(* IEC 61131-3 sources: plc_simulator/services/codesys/POUs (part 11) *)

(* ---- TWA_FB_CalcLimits.st ---- *)
(* ===========================================================================================
 *  TWA_FB_CalcLimits — Transporter Working Area: X-limit calculation
 *
 *  Company : Galvatek part of the John Cockerill Group
 *  Author  : Jarmo Piipponen
 *  Created : 25.03.2026
 *
 * -------------------------------------------------------------------------------------------
 *  Calculates x_min_limit and x_max_limit for all active
 *  transporters. Collision avoidance layers:
 *
 *  Pass 1 (per transporter):
 *  - Station restrictions from g_avoid_status
 *  - Safety distance from same-line neighbors
 *  - canEvade, priority, x-rank computation
 *
 *  Pass 2 (pair comparisons):
 *  - Priority-based restrictions (higher → lower)
 *  - Bidirectional safety (same direction chase)
 *
 *  Final: Trap validation
 *
 *  ------------------------------------------------------------------------------------------
 *
 *  Changes:
 *
 *
 *
 *)

FUNCTION_BLOCK TWA_FB_CalcLimits

(* Introduction of Variables ----------------------------------------------------------------*)

VAR_EXTERNAL CONSTANT
    MAX_TRANSPORTERS        : INT;
    MAX_UNITS               : INT;
    MIN_STATION_INDEX        : INT;
    MAX_STATION_INDEX        : INT;
    AVOID_PASSABLE          : INT;
    AVOID_BLOCK             : INT;
    MIN_WORKING_AREA         : DINT;
    IN_PROCESS              : INT;
END_VAR

VAR_EXTERNAL
  Transporters                     : ARRAY[0..MAX_TRANSPORTERS] OF UDT_TransporterType;
  g_transporter             : ARRAY[1..MAX_TRANSPORTERS] OF UDT_TransporterStatusType;
  Stations                 : ARRAY[MIN_STATION_INDEX..MAX_STATION_INDEX] OF UDT_StationType;
  CountStations              : INT;
  g_avoid_status            : ARRAY[MIN_STATION_INDEX..MAX_STATION_INDEX] OF INT;
  g_station_occupancy             : ARRAY[1..MAX_STATION_INDEX] OF UDT_JC_UnitAtStationType;
  g_batch                   : ARRAY[1..MAX_UNITS] OF UDT_BatchType;
END_VAR

VAR
  i                         : INT;
  j                         : INT;
  stn_num                   : INT;
  stn_x                     : DINT;
  avoid_st                  : INT;
  min_x                     : DINT;
  max_x                     : DINT;
  current_x                 : DINT;
  current_y                 : DINT;
  avoid_dist                : DINT;
  is_target                 : BOOL;
  new_val                   : DINT;

  (* Station scan: nearest restricting station per side *)
  near_left_x               : DINT;
  near_left_stn             : INT;
  near_right_x              : DINT;
  near_right_stn            : INT;
  has_left                  : BOOL;
  has_right                 : BOOL;
  midpoint                  : DINT;

  (* Per-transporter computed values *)
  priority                  : ARRAY[1..MAX_TRANSPORTERS] OF DINT;
  can_evade                 : ARRAY[1..MAX_TRANSPORTERS] OF BOOL;
  rank                      : ARRAY[1..MAX_TRANSPORTERS] OF INT;

  (* Pair comparison *)
  other_x                   : DINT;
  other_y                   : DINT;
  i_phase                   : INT;
  j_phase                   : INT;
  dist                      : DINT;
  work_area                 : DINT;
  a_wins                    : BOOL;
  restrict_x                : DINT;
  between                   : INT;
  chain_ofs                 : DINT;
  adjusted                  : DINT;

  (* Bidirectional *)
  i_moving_right            : BOOL;
  i_moving_left             : BOOL;
  j_moving_right            : BOOL;
  j_moving_left             : BOOL;

  (* IN_PROCESS batch priority boost *)
  lift_stn                  : INT;
  lift_uid                  : INT;
  batch_boost               : DINT;

  (* Full task extent for restrict_x *)
  lift_x                    : DINT;
  sink_x                    : DINT;
  i_lift_stn                : INT;
  i_sink_stn                : INT;
END_VAR

(* ══════════════════════════════════════════════════════════════
   PASS 1: Station restrictions + safety distance + properties
   Each transporter computes its OWN limits in one iteration.
   ══════════════════════════════════════════════════════════════ *)
FOR i := 1 TO MAX_TRANSPORTERS DO
  IF NOT g_transporter[i].IsActive THEN
    priority[i] := 0;
    can_evade[i] := FALSE;
    rank[i] := 0;
    CONTINUE;
  END_IF;

  min_x := Transporters[i].DrivePosMin;
  max_x := Transporters[i].DrivePosMax;
  current_x := g_transporter[i].XPosition;
  current_y := g_transporter[i].YPosition;
  avoid_dist := Transporters[i].AvoidanceWidth;

  (* Lock transporters with no drive range configured *)
  IF (min_x < 1) OR (max_x < 1) THEN
    g_transporter[i].XMinDriveLimit := current_x;
    g_transporter[i].XMaxDriveLimit := current_x;
    priority[i] := 0;
    can_evade[i] := FALSE;
    rank[i] := 0;
    CONTINUE;
  END_IF;

  (* ── Station scan: find nearest restrict LEFT and RIGHT ──────
     Single pass through all stations. Only Block and
     Passable-target stations cause restrictions. *)
  has_left := FALSE;
  has_right := FALSE;
  near_left_x := 0;
  near_left_stn := 0;
  near_right_x := 0;
  near_right_stn := 0;

  FOR stn_num := MIN_STATION_INDEX TO MAX_STATION_INDEX DO
    IF Stations[stn_num].TankId = 0 THEN CONTINUE; END_IF;

    avoid_st := g_avoid_status[stn_num];
    IF avoid_st = 0 THEN CONTINUE; END_IF;  (* AVOID_NONE *)

    (* Passable: only restricts if this transporter's target *)
    IF avoid_st = AVOID_PASSABLE THEN
      is_target := (stn_num = g_transporter[i].LiftStationTarget)
               OR  (stn_num = g_transporter[i].SinkStationTarget);
      IF NOT is_target THEN CONTINUE; END_IF;
    END_IF;

    (* Station is Block or Passable+target → track nearest per side *)
    stn_x := Stations[stn_num].XPosition;

    IF stn_x < current_x THEN
      IF NOT has_left OR stn_x > near_left_x THEN
        near_left_x := stn_x;
        near_left_stn := stn_num;
        has_left := TRUE;
      END_IF;
    ELSIF stn_x > current_x THEN
      IF NOT has_right OR stn_x < near_right_x THEN
        near_right_x := stn_x;
        near_right_stn := stn_num;
        has_right := TRUE;
      END_IF;
    END_IF;
  END_FOR;

  (* Apply station restrictions using station-specific AvoidDistance *)
  IF has_left THEN
    new_val := near_left_x + Stations[near_left_stn].AvoidDistance;
    IF new_val > min_x THEN min_x := new_val; END_IF;
  END_IF;
  IF has_right THEN
    new_val := near_right_x - Stations[near_right_stn].AvoidDistance;
    IF new_val < max_x THEN max_x := new_val; END_IF;
  END_IF;

  (* Conflict: trapped between two restricting stations *)
  IF (min_x >= max_x) AND has_left AND has_right THEN
    midpoint := (near_left_x + near_right_x) / 2;
    min_x := midpoint - 5;
    max_x := midpoint + 5;
  END_IF;

  (* ── Safety distance: each same-line neighbor pushes i away ── *)
  FOR j := 1 TO MAX_TRANSPORTERS DO
    IF j = i THEN CONTINUE; END_IF;
    IF NOT g_transporter[j].IsActive THEN CONTINUE; END_IF;

    other_y := g_transporter[j].YPosition;
    IF ABS(other_y - current_y) >= 1 THEN CONTINUE; END_IF;

    other_x := g_transporter[j].XPosition;

    IF other_x < current_x THEN
      (* j is LEFT → j's safety zone pushes i's min up *)
      new_val := other_x + Transporters[j].AvoidanceWidth;
  IF new_val > min_x THEN min_x := new_val; END_IF;
    ELSIF other_x > current_x THEN
      (* j is RIGHT → j's safety zone pushes i's max down *)
      new_val := other_x - Transporters[j].AvoidanceWidth;
  IF new_val < max_x THEN max_x := new_val; END_IF;
    END_IF;
  END_FOR;

  (* ── Write limits ── *)
  g_transporter[i].XMinDriveLimit := min_x;
  g_transporter[i].XMaxDriveLimit := max_x;

  (* ── canEvade (inline) ── *)
  can_evade[i] := TRUE;
  IF g_transporter[i].Status < 3 THEN
    can_evade[i] := FALSE;
  END_IF;
  IF (g_transporter[i].Status = 4)
     AND ((g_transporter[i].Phase = 2) OR (g_transporter[i].Phase = 4)) THEN
    can_evade[i] := FALSE;
  END_IF;
  work_area := max_x - min_x;
  IF work_area < MIN_WORKING_AREA THEN
    can_evade[i] := FALSE;
  END_IF;

  (* ── Priority (inline, replaces TWA_CalcPriority call) ──────
     IN_PROCESS batch boost: +100000 if the task serves an
     IN_PROCESS batch. Phases 1-4 all check via LiftStation
     unit lookup (unit stays associated throughout transfer).
     This ensures treatment tasks trump NTT/empty moves. ── *)
  i_phase := g_transporter[i].Phase;
  batch_boost := 0;
  IF i_phase >= 1 AND i_phase <= 4 THEN
    lift_stn := g_transporter[i].LiftStationTarget;
    IF lift_stn >= 1 AND lift_stn <= MAX_STATION_INDEX THEN
      lift_uid := g_station_occupancy[lift_stn].UnitId;
      IF lift_uid >= 1 AND lift_uid <= MAX_UNITS THEN
        IF g_batch[lift_uid].State = IN_PROCESS THEN
          batch_boost := DINT#100000;
        END_IF;
      END_IF;
    END_IF;
  END_IF;

  IF NOT can_evade[i] THEN
    priority[i] := DINT#100000;
  ELSIF i_phase = 3 OR i_phase = 4 THEN
    dist := ABS(current_x - g_transporter[i].XFinalTarget);
  IF dist > 99999 THEN dist := 99999; END_IF;
    priority[i] := DINT#200000 + batch_boost + (DINT#99999 - dist);
  ELSIF i_phase = 1 OR i_phase = 2 THEN
    (* Move-away (Status=3, Phase=1) gets idle-class priority, not active-task priority *)
    IF g_transporter[i].Status = 3 THEN
      priority[i] := 2;  (* above stationary idle (1), below active tasks (100000+) *)
    ELSE
      dist := ABS(current_x - g_transporter[i].XFinalTarget);
      IF dist > 99999 THEN dist := 99999; END_IF;
      priority[i] := DINT#100000 + batch_boost + (DINT#99999 - dist);
    END_IF;
  ELSE
    priority[i] := 1;
  END_IF;

  (* ── X-rank among same-line active transporters ──
     rank = 1 + count of same-line transporters with smaller x *)
  rank[i] := 1;
  FOR j := 1 TO MAX_TRANSPORTERS DO
    IF j = i THEN CONTINUE; END_IF;
    IF NOT g_transporter[j].IsActive THEN CONTINUE; END_IF;
    IF ABS(g_transporter[j].YPosition - current_y) >= 1 THEN CONTINUE; END_IF;
    IF g_transporter[j].XPosition < current_x THEN
      rank[i] := rank[i] + 1;
    END_IF;
  END_FOR;
END_FOR;

(* ══════════════════════════════════════════════════════════════
   PASS 2: Priority restrictions + bidirectional safety
   Each pair (i,j): i restricts j if i has higher priority.
   ══════════════════════════════════════════════════════════════ *)
FOR i := 1 TO MAX_TRANSPORTERS DO
  IF NOT g_transporter[i].IsActive THEN CONTINUE; END_IF;
  IF priority[i] = 0 THEN CONTINUE; END_IF;

  current_x := g_transporter[i].XPosition;
  current_y := g_transporter[i].YPosition;
  i_phase := g_transporter[i].Phase;

  FOR j := 1 TO MAX_TRANSPORTERS DO
    IF j = i THEN CONTINUE; END_IF;
    IF NOT g_transporter[j].IsActive THEN CONTINUE; END_IF;
    IF priority[j] = 0 THEN CONTINUE; END_IF;

    other_y := g_transporter[j].YPosition;
    IF ABS(other_y - current_y) >= 1 THEN CONTINUE; END_IF;

    other_x := g_transporter[j].XPosition;
    j_phase := g_transporter[j].Phase;

    (* ── Priority restrictions: i restricts j if i wins ── *)
    (* Move-away (Status=3, Phase=1) participates in restrictions
       so it can push stationary idle transporters out of its way *)
    IF (i_phase <> 0) OR (g_transporter[i].Status = 3 AND i_phase = 1) THEN
      a_wins := FALSE;
      IF priority[i] > priority[j] THEN
        a_wins := TRUE;
      ELSIF (priority[i] = priority[j]) AND (i < j) THEN
        a_wins := TRUE;
      END_IF;

      IF a_wins THEN
        (* Full task extent: use the extreme position
           of both lift and sink stations on the side
           facing j. This prevents j from first driving
           closer and then having to reverse when i
           moves to the other end of its task. *)
        i_lift_stn := g_transporter[i].LiftStationTarget;
        i_sink_stn := g_transporter[i].SinkStationTarget;
        IF i_phase >= 1 AND i_phase <= 4 THEN
          lift_x := current_x;
          sink_x := current_x;
          IF i_lift_stn >= MIN_STATION_INDEX
             AND i_lift_stn <= MAX_STATION_INDEX THEN
            lift_x := Stations[i_lift_stn].XPosition;
          END_IF;
          IF i_sink_stn >= MIN_STATION_INDEX
             AND i_sink_stn <= MAX_STATION_INDEX THEN
            sink_x := Stations[i_sink_stn].XPosition;
          END_IF;
          IF current_x < other_x THEN
            (* i LEFT of j → use rightmost extent *)
            restrict_x := lift_x;
            IF sink_x > restrict_x THEN
              restrict_x := sink_x;
            END_IF;
            IF current_x > restrict_x THEN
              restrict_x := current_x;
            END_IF;
          ELSE
            (* i RIGHT of j → use leftmost extent *)
            restrict_x := lift_x;
            IF sink_x < restrict_x THEN
              restrict_x := sink_x;
            END_IF;
            IF current_x < restrict_x THEN
              restrict_x := current_x;
            END_IF;
          END_IF;
        ELSE
          restrict_x := current_x;
        END_IF;

        (* "between" from pre-computed rank *)
        between := ABS(rank[i] - rank[j]) - 1;
  IF between < 0 THEN between := 0; END_IF;

        chain_ofs := Transporters[i].AvoidanceWidth
                   + INT_TO_DINT(between) * (MIN_WORKING_AREA + Transporters[i].AvoidanceWidth);

        IF current_x < other_x THEN
          (* i LEFT, j RIGHT → restrict j's XMin *)
          new_val := restrict_x + chain_ofs;
          IF new_val > g_transporter[j].XMinDriveLimit THEN
            IF new_val <= (g_transporter[j].XMaxDriveLimit - MIN_WORKING_AREA) THEN
              g_transporter[j].XMinDriveLimit := new_val;
            ELSE
              adjusted := g_transporter[j].XMaxDriveLimit - MIN_WORKING_AREA;
              IF adjusted > g_transporter[j].XMinDriveLimit THEN
                g_transporter[j].XMinDriveLimit := adjusted;
              END_IF;
            END_IF;
          END_IF;

        ELSIF current_x > other_x THEN
          (* i RIGHT, j LEFT → restrict j's XMax *)
          new_val := restrict_x - chain_ofs;
          IF new_val < g_transporter[j].XMaxDriveLimit THEN
            IF new_val >= (g_transporter[j].XMinDriveLimit + MIN_WORKING_AREA) THEN
              g_transporter[j].XMaxDriveLimit := new_val;
            ELSE
              adjusted := g_transporter[j].XMinDriveLimit + MIN_WORKING_AREA;
              IF adjusted < g_transporter[j].XMaxDriveLimit THEN
                g_transporter[j].XMaxDriveLimit := adjusted;
              END_IF;
            END_IF;
          END_IF;
        END_IF;
      END_IF;
    END_IF;

    (* ── Bidirectional safety: only adjacent (rank diff = 1) ── *)
    IF ABS(rank[i] - rank[j]) = 1 THEN
      i_moving_right := ((i_phase = 1) OR (i_phase = 3))
                        AND (g_transporter[i].XFinalTarget > current_x);
      j_moving_right := ((j_phase = 1) OR (j_phase = 3))
                        AND (g_transporter[j].XFinalTarget > other_x);
      i_moving_left := ((i_phase = 1) OR (i_phase = 3))
                       AND (g_transporter[i].XFinalTarget < current_x);
      j_moving_left := ((j_phase = 1) OR (j_phase = 3))
                       AND (g_transporter[j].XFinalTarget < other_x);

      IF current_x < other_x AND i_moving_right AND j_moving_right THEN
        (* i LEFT chasing j RIGHT → restrict j's XMin *)
        new_val := current_x + Transporters[i].AvoidanceWidth;
        IF new_val > g_transporter[j].XMinDriveLimit THEN
          g_transporter[j].XMinDriveLimit := new_val;
        END_IF;
      END_IF;

      IF current_x > other_x AND i_moving_left AND j_moving_left THEN
        (* i RIGHT chasing j LEFT → restrict j's XMax *)
        new_val := current_x - Transporters[i].AvoidanceWidth;
        IF new_val < g_transporter[j].XMaxDriveLimit THEN
          g_transporter[j].XMaxDriveLimit := new_val;
        END_IF;
      END_IF;
    END_IF;
  END_FOR;
END_FOR;

(* ══════════════════════════════════════════════════════════════
   TRAP VALIDATION: if restrictions conflict, lock in place
   ══════════════════════════════════════════════════════════════ *)
FOR i := 1 TO MAX_TRANSPORTERS DO
  IF NOT g_transporter[i].IsActive THEN CONTINUE; END_IF;
  IF g_transporter[i].XMinDriveLimit > g_transporter[i].XMaxDriveLimit THEN
    g_transporter[i].XMinDriveLimit := g_transporter[i].XPosition;
    g_transporter[i].XMaxDriveLimit := g_transporter[i].XPosition;
  END_IF;
END_FOR;

END_FUNCTION_BLOCK

(* ---- Main.st ---- *)
(* ===========================================================================================
 *  Main — Main program (CODESYS / OPC UA)
 *
 *  Company : Galvatek part of the John Cockerill Group
 *  Author  : Jarmo Piipponen
 *  Created : 25.03.2026
 *
 * -------------------------------------------------------------------------------------------
 *  Simulator version: delegates SIM-specific logic to FB_SIM_MainCycle.
 *
 *  Production version would replace sim_main with:
 *    - Real PLC clock → g_time_s
 *    - TWA calc
 *    - (no command handler, no physics, no UI snapshot, no event queue)
 *
 *  ------------------------------------------------------------------------------------------
 *
 *  Changes:
 *
 *
 *
 *)

PROGRAM Main

(* Introduction of Variables ----------------------------------------------------------------*)

VAR_EXTERNAL
  g_time_s                  : LINT;
END_VAR

VAR
  sim_main                  : FB_SIM_MainCycle;
  main_scheduler            : FB_STC_MainScheduler;
END_VAR

(* ── Simulator: command handler, time, TWA, physics, UI snapshot, events ── *)
sim_main();

(* ── Main Scheduler (TSK + DEP alternating cycles) ──
   MUST run outside init_done block so that when init_done=FALSE
   (during RESET), MainScheduler's i_run=FALSE path executes,
   properly resetting internal state of both TSK and DEP FBs. *)
main_scheduler(i_run := sim_main.o_init_done, i_time_s := g_time_s);

END_PROGRAM

(* ---- plc_prg.st ---- *)
(* ============================================================
   plc_prg.st — Main program (CODESYS / OPC UA)
   ============================================================
   Gateway communicates via OPC UA — reads/writes GVL variables
   directly. All multi-field writes are atomic (single OPC UA call).

   Gateway writes:
     g_station[], g_cfg[], g_unit[], g_batch[], g_program[],
     g_ntt[], g_cal[], g_avoid_status[], g_time_s,
     g_production_queue, g_event_ack_seq

   Gateway reads:
     g_transporter[], g_schedule[], g_task[], g_sim_trans[],
     g_move[], g_event, g_dep_wait_sched, g_sched_dbg_*,
     g_cal_active, g_cal[]

   Command interface (g_cmd_code / g_cmd_param):
     Gateway writes g_cmd_code + g_cmd_param via OPC UA.
     PLC processes when g_cmd_code <> 0, then clears it.
     2 = init       (param = station_count)
     3 = clear      (clear all config)
     8 = cal_ctrl   (param: 1=start, 2=calculate, 3=abort)
    12 = calc_move  (compute g_move from g_cal kinematics)
   ============================================================ *)

PROGRAM PLC_PRG
VAR_EXTERNAL CONSTANT
    MAX_Transporters    : INT;
    MAX_STATIONS_PER_STEP : INT;
    MIN_StationIndex    : INT;
    MAX_StationIndex    : INT;
    MAX_Units           : INT;
    DEP_MAX_WAITING     : INT;
END_VAR

VAR_EXTERNAL
  (* --- Shared data arrays — written by Gateway via OPC UA --- *)
  g_station_count    : INT;
  g_station          : ARRAY[MIN_StationIndex..MAX_StationIndex] OF UDT_StationType;
  g_station_loc      : ARRAY[1..MAX_StationIndex] OF UDT_UnitLocation;
  g_cfg              : ARRAY[1..MAX_Transporters] OF UDT_TransporterType;
  g_transporter      : ARRAY[1..MAX_Transporters] OF UDT_TransporterStatusType;
  g_sim_trans        : ARRAY[1..MAX_Transporters] OF UDT_JC_SimTransporterType;
  g_unit             : ARRAY[1..MAX_Units] OF UDT_UnitType;
  g_ntt              : ARRAY[1..MAX_Transporters] OF UDT_JC_NttTransporterType;
  g_batch            : ARRAY[1..MAX_Units] OF UDT_BatchType;
  g_program          : ARRAY[1..MAX_Units] OF UDT_TreatmentProgramType;
  g_avoid_status     : ARRAY[MIN_StationIndex..MAX_StationIndex] OF INT;
  g_move             : ARRAY[1..MAX_Transporters] OF UDT_JC_MoveTimesType;
  g_schedule         : ARRAY[1..MAX_Units] OF UDT_JC_TskScheduleType;
  g_task             : ARRAY[1..MAX_Transporters] OF UDT_JC_TskQueueType;
  (* --- Departure Scheduler state --- *)
  g_dep_activated    : BOOL;
  g_dep_stable       : BOOL;
  g_dep_waiting_count : INT;
  g_dep_overlap      : UDT_JC_DepOverlapType;
  g_dep_pending      : UDT_JC_DepPendingWriteType;
  g_dep_waiting      : ARRAY[1..DEP_MAX_WAITING] OF INT;
  g_dep_wait_sched   : UDT_JC_TskScheduleType;
  g_dep_wait_unit    : INT;
  (* --- Scheduler Debug --- *)
  g_sched_dbg_tsk_phase : INT;
  g_sched_dbg_dep_phase : INT;
  g_sched_dbg_turn      : INT;
  g_conflict_resolved   : BOOL;
  g_sched_dbg_batch_cnt : INT;
  (* --- Calibration --- *)
  g_cal              : ARRAY[1..MAX_Transporters] OF UDT_JC_CalibrationType;
  g_cal_active       : BOOL;
  (* --- Production --- *)
  g_production_queue : INT;
  (* --- Time --- *)
  g_time_s           : LINT;
  (* --- Event queue --- *)
  g_event            : UDT_JC_EventQueueType;
  g_event_pending    : UDT_JC_EventMsgType;
  g_event_pending_valid : BOOL;
  g_event_ack_seq    : INT;
  (* --- OPC UA Command Interface --- *)
  g_cmd_code         : INT;
  g_cmd_param        : INT;
END_VAR

VAR
  init_done      : BOOL := FALSE;
  i              : INT;
  twa_calc       : TWA_FB_CalcLimits;
  clear_cfg      : SIM_FB_ClearConfig;
  cycle_count    : INT;
  main_sched     : STC_FB_MainScheduler;
  run_tasks      : SIM_FB_RunTasks;
  calibrate      : STC_FB_Calibrate;
  calc_move      : STC_FB_CalcMoveTimes;
  evt_queue      : STC_FB_EventQueue;
  cal_cmd        : INT := 0;
  cal_load_run   : BOOL := FALSE;
  (* Time self-increment *)
  time_cycle_cnt : INT := 0;
  last_time_s    : LINT := 0;
  (* Waiting batch at station 114 *)
  fb_wait_calc       : TSK_FB_CalcSchedule;
  dep_wait_114_unit  : INT := 0;
  dep_wait_114_last  : INT := 0;
  wait_i             : INT;
END_VAR

(* ============================================================
   COMMAND HANDLER — OPC UA (direct, no sequence handshake)
   Gateway writes g_cmd_code + g_cmd_param in one atomic OPC UA
   call. PLC processes when g_cmd_code <> 0 and clears it.
   ============================================================ *)
IF g_cmd_code <> 0 THEN

  IF g_cmd_code = 3 THEN
    (* ── Clear all config data ── *)
    clear_cfg();
    init_done := FALSE;
    g_station_count := 0;

  ELSIF g_cmd_code = 8 THEN
    (* ── Calibration control ── *)
    cal_cmd := g_cmd_param;

  ELSIF g_cmd_code = 12 THEN
    (* ── Compute g_move from loaded g_cal kinematic params ── *)
    cal_load_run := TRUE;

  ELSIF g_cmd_code = 2 THEN
    (* ── Finish init: all config already uploaded via OPC UA ── *)
    g_station_count := g_cmd_param;

    FOR i := 1 TO MAX_Transporters DO
      IF g_cfg[i].TaskArea[1].MinLift > 0 THEN
        g_transporter[i].IsActive := TRUE;
        g_transporter[i].Status := 3;  (* auto_idle *)
      ELSE
        g_transporter[i].IsActive := FALSE;
        g_transporter[i].Status := 0;  (* not_used *)
      END_IF;
      g_transporter[i].Phase := 0;
      g_sim_trans[i].ZStage := 0;
      g_sim_trans[i].XVelocity := 0;
      g_sim_trans[i].ZTimer := 0.0;
      g_transporter[i].XMinDriveLimit := g_cfg[i].DrivePosMin;
      g_transporter[i].XMaxDriveLimit := g_cfg[i].DrivePosMax;

      (* Start position: at own area minimum, z=0 *)
      g_transporter[i].XPosition := g_cfg[i].DrivePosMin;
      g_transporter[i].ZPosition := 0;
      g_transporter[i].CurrentStation := 0;
    END_FOR;

    init_done := TRUE;

    (* Init event queue *)
    g_event.Head := 1;
    g_event.NextSeq := 1;
    g_event.Count := 0;
  END_IF;

  g_cmd_code := 0;  (* Command processed — clear trigger *)
END_IF;

(* ============================================================
   MAIN TRANSPORT CYCLE — only runs when init_done
   ============================================================ *)
IF init_done THEN

  (* ── Compute g_move from loaded kinematic params (one-shot) ── *)
  calc_move(i_run := cal_load_run);
  IF cal_load_run THEN
    cal_load_run := FALSE;
  END_IF;

  (* ── Calculate transporter working areas (X-limits) every cycle ── *)
  twa_calc();

  (* ── Unix time self-increment ──
     Gateway writes g_time_s directly via OPC UA for sync.
     PLC self-increments +1 second every 50 cycles (50 × 20 ms = 1 s)
     when gateway hasn't updated. *)
  IF g_time_s <> last_time_s THEN
    (* Gateway wrote new time — accept and reset counter *)
    last_time_s := g_time_s;
    time_cycle_cnt := 0;
  ELSE
    time_cycle_cnt := time_cycle_cnt + 1;
    IF time_cycle_cnt >= 50 THEN
      g_time_s := g_time_s + LINT#1;
      last_time_s := g_time_s;
      time_cycle_cnt := 0;
    END_IF;
  END_IF;

  (* ── Execute transporter tasks (physics simulation) ── *)
  run_tasks(i_run := init_done);

  (* ── Calibration FB — issues test tasks, measures parameters ── *)
  calibrate(i_run := init_done, i_cmd := cal_cmd);
  cal_cmd := 0;
  g_cal_active := calibrate.o_active;

END_IF;  (* init_done *)

(* ── Main Scheduler (TSK + DEP alternating cycles) ──
   MUST run outside init_done block so that when init_done=FALSE
   (during RESET), MainScheduler's i_run=FALSE path executes,
   properly resetting internal state of both TSK and DEP FBs. *)
main_sched(i_run := init_done, i_time_s := g_time_s);

(* ── Event queue — always runs, not gated by init_done ── *)
evt_queue();

(* ── Cycle counter ── *)
cycle_count := cycle_count + 1;
IF cycle_count > 30000 THEN cycle_count := 0; END_IF;

(* ── WAITING BATCH AT STATION 114 — shortcut for UI ──
   Scan for NOT_PROCESSED unit at station 114 with valid program.
   Calculate schedule once when a new unit appears there. *)
dep_wait_114_unit := 0;
FOR wait_i := 1 TO 10 DO
  IF g_unit[wait_i].location = 114
     AND g_batch[wait_i].State = 0
     AND g_program[wait_i].ProgramId > 0
     AND g_batch[wait_i].ProgId = g_program[wait_i].ProgramId THEN
    dep_wait_114_unit := wait_i;
  END_IF;
END_FOR;

IF dep_wait_114_unit <> dep_wait_114_last THEN
  dep_wait_114_last := dep_wait_114_unit;
  IF dep_wait_114_unit > 0 THEN
    fb_wait_calc(i_unit := dep_wait_114_unit, i_trans := 1, i_time_s := g_time_s);
    g_dep_wait_sched := g_schedule[dep_wait_114_unit];
    g_dep_wait_unit  := dep_wait_114_unit;
    g_schedule[dep_wait_114_unit].StageCount := 0;
  ELSE
    g_dep_wait_unit := 0;
  END_IF;
END_IF;

END_PROGRAM
